FUNCTION_BLOCK MotorDC (* Service Interface Function Block Type *)
  (* Standard: 61499-2 *)
  (* Version 0.0, 2012-05-20, 4DIAC-IDE, 4DIAC-Consortium *)
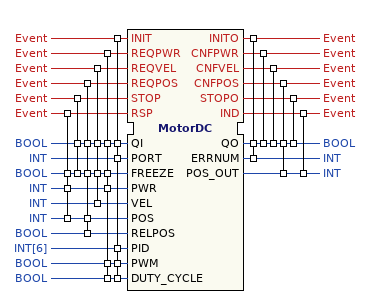
  EVENT_INPUT
    INIT WITH PORT, PID, QI, DUTY_CYCLE, PWM; (* Service Initialization *)
    REQPWR WITH PWR, FREEZE, PWM, DUTY_CYCLE, QI; (* Service Request *)
    REQVEL WITH FREEZE, VEL, QI; (* move with velocity request *)
    REQPOS WITH POS, FREEZE, RELPOS, QI; (* move to position request *)
    STOP WITH QI, FREEZE; (* stop motor *)
    RSP WITH FREEZE, PWR, POS; (* Returns whether the motor has finished a move with specified position. *)
  END_EVENT
  EVENT_OUTPUT
    INITO WITH QO, ERRNUM; (* Initialization Confirm *)
    CNFPWR WITH QO; (* Confirmation of Requested Service *)
    CNFVEL WITH QO;
    CNFPOS WITH POS_OUT, QO;
    STOPO WITH QO; (* stop confirmation *)
    IND WITH POS_OUT; (* specified position.reached *)
  END_EVENT
  VAR_INPUT
    QI : BOOL; (* input qualifer *)
    PORT : INT; (* Port the Motor is connected *)
    FREEZE : BOOL; (* when turn off then true freeze; false coast *)
    PWR : INT; (* 100 (full forward) to -100 (full backward) *)
    VEL : INT; (* -1000 to 1000 ticks per second. *)
    POS : INT; (* -1000 to 1000 ticks per second *)
    RELPOS : BOOL; (* Relative position = true; Absolute position = false *)
    PID : ARRAY [0..5] OF INT; (* [P,I,D,PD,ID,DD] default is {30,0,-30,70,1,51} *)
    PWM : BOOL; (* true = use PWM *)
    DUTY_CYCLE : BOOL; (* PWM  proportion of 'on' time to the regular interval or 'period' of time; *)
  END_VAR
  VAR_OUTPUT
    QO : BOOL; (* Event Output Qualifier; false if Port problem *)
    ERRNUM : INT; (* error number 1=port error; 2=postion error *)
    POS_OUT : INT;
  END_VAR
  SERVICE APPLICATION/RESOURCE (* Service Interface Function Block Type *)
    SEQUENCE normal_establishment
      APPLICATION.INIT+(PARAMS) -> APPLICATION.INITO+(PARAMS);
    END_SEQUENCE
    SEQUENCE unsuccessful_establishment
      APPLICATION.INIT+(PARAMS) -> APPLICATION.INITO-(STATUS);
    END_SEQUENCE
    SEQUENCE request_confirm
      APPLICATION.REQ+(SD) -> APPLICATION.CNF+(RD);
    END_SEQUENCE
    SEQUENCE request_inhibited
      APPLICATION.REQ-(SD) -> APPLICATION.CNF-(STATUS);
    END_SEQUENCE
    SEQUENCE request_error
      APPLICATION.REQ+(SD) -> APPLICATION.CNF-(STATUS);
    END_SEQUENCE
    SEQUENCE indication_response
      RESOURCE.indicate(RD) -> APPLICATION.IND+(RD);
      APPLICATION.RSP(QI,SD) -> RESOURCE.response(QI,SD);
    END_SEQUENCE
    SEQUENCE indication_inhibited
      RESOURCE.indicate(RD,QI=FALSE) -> RESOURCE.inhibited();
    END_SEQUENCE
    SEQUENCE error_indication
      RESOURCE.error(STATUS) -> APPLICATION.IND-(STATUS);
    END_SEQUENCE
    SEQUENCE application_initiated_termination
      APPLICATION.INIT-() -> APPLICATION.INITO-(STATUS);
    END_SEQUENCE
    SEQUENCE resource_initiated_termination
      -> APPLICATION.INITO-(STATUS);
    END_SEQUENCE
  END_SERVICE
END_FUNCTION_BLOCK
